// TwinCAT 3 PLC project IotMqttSampleAzureIotSuitePlc
// ProgramVersion: 3.1.4021.2
// libraries:
//   Tc2_Standard, * (Beckhoff Automation GmbH)
//   Tc2_System, * (Beckhoff Automation GmbH)
//   Tc3_IotBase, * (Beckhoff Automation GmbH)
//   Tc3_JsonXml, * (Beckhoff Automation GmbH)
//   Tc3_Module, * (Beckhoff Automation GmbH)
// project tree:
//   DUTs/ ST_Values.TcDUT
//   GVLs/ GVL.TcGVL (not stored)
//   / PlcTask.TcTTO (not stored)
//   POUs/HelperFunctions/DeviceTwin/ F_DeviceTwin_GetSubscriberTopicStatusCodes.TcPOU (not stored), F_DeviceTwin_GetSubscriberTopicDesired.TcPOU, F_DeviceTwin_GetPublisherTopic.TcPOU, F_DeviceTwin_GetReportedProperties.TcPOU, F_DeviceTwin_IsDesiredTopic.TcPOU
//   POUs/HelperFunctions/ F_GenerateData.TcPOU (not stored), F_GetPublisherTopic.TcPOU
//   POUs/ MAIN.TcPOU (not stored), PrgMqttCom.TcPOU (not stored)
// real-time tasks:
//   TASK PlcTask: cycle T#10ms, priority 20, ADS port 350

// ---- DUTs/ST_Values.TcDUT
TYPE ST_Values :
STRUCT
	  {attribute 'Unit' := 'm/s'}
	  {attribute 'DisplayName' := 'Speed'}
	  Sensor1   : REAL := 42.42;
	  {attribute 'Unit' := 'V'}
	  {attribute 'DisplayName' := 'Voltage'}
	  Sensor2	: DINT := 230;
	  {attribute 'Unit' := 'A'}
	  {attribute 'DisplayName' := 'Current'}
	  Sensor3	: DINT := 3;
END_STRUCT
END_TYPE

// ---- POUs/HelperFunctions/DeviceTwin/F_DeviceTwin_GetSubscriberTopicDesired.TcPOU
FUNCTION F_DeviceTwin_GetSubscriberTopicDesired : STRING
VAR_INPUT
END_VAR
VAR
END_VAR

F_DeviceTwin_GetSubscriberTopicDesired := '$$iothub/twin/PATCH/properties/desired/#';

END_FUNCTION

// ---- POUs/HelperFunctions/DeviceTwin/F_DeviceTwin_GetPublisherTopic.TcPOU
FUNCTION F_DeviceTwin_GetPublisherTopic : STRING
VAR_INPUT
END_VAR
VAR
END_VAR

F_DeviceTwin_GetPublisherTopic := '$$iothub/twin/PATCH/properties/reported/?$rid=42';

END_FUNCTION

// ---- POUs/HelperFunctions/DeviceTwin/F_DeviceTwin_GetReportedProperties.TcPOU
FUNCTION F_DeviceTwin_GetReportedProperties : STRING(2000)
VAR_INPUT
END_VAR
VAR
	(* JSON document *)
	fbJsonDeviceInfo 	: FB_JsonSaxWriter;
	sJsonDocDeviceInfo 	: STRING(2000);
END_VAR

fbJsonDeviceInfo.StartObject();
fbJsonDeviceInfo.AddKey('Device');
fbJsonDeviceInfo.StartObject();
fbJsonDeviceInfo.AddKey('Location');
fbJsonDeviceInfo.StartObject();
fbJsonDeviceInfo.AddKey('Latitude');
fbJsonDeviceInfo.AddString('51.881034');
fbJsonDeviceInfo.AddKey('Longitude');
fbJsonDeviceInfo.AddString('8.491037');
fbJsonDeviceInfo.EndObject();
fbJsonDeviceInfo.EndObject();
fbJsonDeviceInfo.AddKey('System');
fbJsonDeviceInfo.StartObject();
fbJsonDeviceInfo.AddKey('Manufacturer');
fbJsonDeviceInfo.AddString('Beckhoff Automation');
fbJsonDeviceInfo.AddKey('Firmware');
fbJsonDeviceInfo.AddString('1.42');
fbJsonDeviceInfo.AddKey('InstalledRAM');
fbJsonDeviceInfo.AddString('4 GB');
fbJsonDeviceInfo.AddKey('Processor');
fbJsonDeviceInfo.AddString('Intel Core i5');
fbJsonDeviceInfo.EndObject();
fbJsonDeviceInfo.EndObject();
sJsonDocDeviceInfo := fbJsonDeviceInfo.GetDocument();
F_DeviceTwin_GetReportedProperties := sJsonDocDeviceInfo;

END_FUNCTION

// ---- POUs/HelperFunctions/DeviceTwin/F_DeviceTwin_IsDesiredTopic.TcPOU
FUNCTION F_DeviceTwin_IsDesiredTopic : BOOL
VAR_INPUT
	sTopic : STRING; // $iothub/twin/PATCH/properties/desired/#	  
END_VAR
VAR
END_VAR

IF FIND(sTopic, '$$iothub/twin/PATCH/properties/desired/') = 0 THEN
	  F_DeviceTwin_IsDesiredTopic := FALSE;
ELSE
	  F_DeviceTwin_IsDesiredTopic := TRUE;
END_IF

END_FUNCTION

// ---- POUs/HelperFunctions/F_GetPublisherTopic.TcPOU
FUNCTION F_GetPublisherTopic : STRING(255)
VAR_INPUT
	  sDeviceId			: STRING;
END_VAR
VAR
	  sPublisherTopic 	: STRING;
	  sTopicFirst 		: STRING := 'devices/';
	  sTopicSecond		: STRING := '/messages/events/readpipe/';
END_VAR

sPublisherTopic := CONCAT(sTopicFirst, sDeviceId);
sPublisherTopic := CONCAT(sPublisherTopic, sTopicSecond);
F_GetPublisherTopic := sPublisherTopic;

END_FUNCTION
